PROGRAM Q7
VAR
	 A : BOOL := TRUE;
 B : BOOL := FALSE;
 C : BOOL := FALSE;
END_VAR

// Result: C == TRUE;

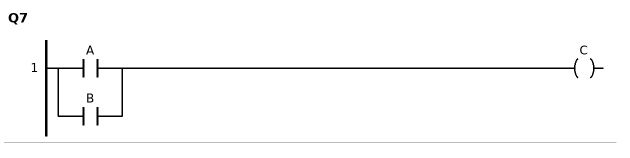
// NETWORK 1
C := A OR B;

END_PROGRAM

(* stored: Version 1.1.0.1, ProductVersion 3.1.4024.12
   POU Q7: Id {730e29e2-cfe0-4de9-812d-8cf9abbb9c6a}, SpecialFunc None *)
